FUNCTION_BLOCK IN_TEXT (* WSTRING input from TextArea *)
  (* Standard: 61499-1; Classification: GUI *)
  (* Version 0.3, 2004-06-20, JHC, Rockwell Automation, Changed semantics of REQ- to clear(). *)
  (* Version 0.2, 2002-05-03, JHC, Rockwell Automation, Made QI IV=true. *)
  (* Version 0.1, 2001-11-26, JHC, Rockwell Automation, Changed ROWS,COLS to SIZE. *)
  (* Version 0.0, 2001-10-09, JHC, Rockwell Automation, Copied/Modified from IN_ANY *)
  (* Compiler header: package fb.rt.hmi.*; *)
  (* Compiler Java IBM VisualAge 3.0 *)
  (* Compiler Java IBM Jikes 1.0.6 *)
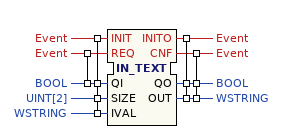
  EVENT_INPUT
    INIT WITH QI, SIZE, IVAL;
    REQ WITH QI;
  END_EVENT
  EVENT_OUTPUT
    INITO WITH QO, OUT;
    CNF WITH QO, OUT;
  END_EVENT
  VAR_INPUT
    QI : BOOL := true;
    SIZE : ARRAY [0..1] OF UINT := [10,50]; (* [rows,columns] *)
    IVAL : WSTRING;
  END_VAR
  VAR_OUTPUT
    QO : BOOL; (* 1=OK,0=Error *)
    OUT : WSTRING;
  END_VAR
  SERVICE IN_TEXT/TextArea
    SEQUENCE normal_initialization
      IN_TEXT.INIT+(IVAL) -> TextArea.initialize(IVAL) -> IN_TEXT.INITO+(OUT);
    END_SEQUENCE
    SEQUENCE initialization_inhibited
      IN_TEXT.INIT-() -> IN_TEXT.INITO-();
    END_SEQUENCE
    SEQUENCE data_request
      IN_TEXT.REQ+() -> TextArea.getText() -> IN_TEXT.CNF+(OUT);
    END_SEQUENCE
    SEQUENCE not_initialized
      IN_TEXT.REQ+() -> IN_TEXT.CNF-();
    END_SEQUENCE
    SEQUENCE clear
      IN_TEXT.REQ-() -> TextArea.clear() -> IN_TEXT.CNF-();
    END_SEQUENCE
  END_SERVICE
END_FUNCTION_BLOCK
